// TIA Portal V20 export
FUNCTION_BLOCK "LER_Axis"   // FB60, LAD
// stored: Access Published, MemoryReserve 100, Namespace Homing, SetENOAutomatically false
   VAR_INPUT
      Status : "LAF_typeUnitStatus";
      HMI : Bool;
      Process : Bool;
      int1 { ExternalAccessible := 'False'; ExternalVisible := 'False'; ExternalWritable := 'False'} : Bool := true;
      int2 { ExternalAccessible := 'False'; ExternalVisible := 'False'; ExternalWritable := 'False'} : Bool := true;
      int3 { ExternalAccessible := 'False'; ExternalVisible := 'False'; ExternalWritable := 'False'} : Bool := true;
      int4 { ExternalAccessible := 'False'; ExternalVisible := 'False'; ExternalWritable := 'False'} : Bool := true;
      int5 { ExternalAccessible := 'False'; ExternalVisible := 'False'; ExternalWritable := 'False'} : Bool := true;
      int6 { ExternalAccessible := 'False'; ExternalVisible := 'False'; ExternalWritable := 'False'} : Bool := true;
      int7 { ExternalAccessible := 'False'; ExternalVisible := 'False'; ExternalWritable := 'False'} : Bool := true;
      int8 { ExternalAccessible := 'False'; ExternalVisible := 'False'; ExternalWritable := 'False'} : Bool := true;
      int9 { ExternalAccessible := 'False'; ExternalVisible := 'False'; ExternalWritable := 'False'} : Bool := true;
      int10 { ExternalAccessible := 'False'; ExternalVisible := 'False'; ExternalWritable := 'False'} : Bool := true;
      Bypass : Bool := true;
   END_VAR
   VAR_OUTPUT
      HomeInterlock : Bool;
   END_VAR
   VAR_IN_OUT
      intout : Array[0..9] of Bool;
   END_VAR
   VAR
      HomeCondition : Bool;
      HomeNotCondition : Bool;
   END_VAR
BEGIN

REGION Network 2 (SCL)
       IF (#int1 AND #int2 AND #int3 AND #int4 AND #int5 AND #int6 AND #int7 AND #int8 AND #int9 AND #int10) OR #Bypass THEN
           #HomeCondition := TRUE;
           #HomeNotCondition := FALSE;


           IF #HMI OR #Process THEN
               #intout[0] := FALSE;
               #intout[1] := FALSE;
               #intout[2] := FALSE;
               #intout[3] := FALSE;
               #intout[4] := FALSE;
               #intout[5] := FALSE;
               #intout[6] := FALSE;
               #intout[7] := FALSE;
               #intout[8] := FALSE;
               #intout[9] := FALSE;
           END_IF;


    ELSE
               #HomeCondition := FALSE;
               #HomeNotCondition := TRUE;

           IF #HMI OR #Process THEN

               IF NOT #int1 THEN
                   #intout[0] := TRUE;
               ELSE
                   #intout[0] := FALSE;
               END_IF;
               IF NOT #int2 THEN
                   #intout[1] := TRUE;
               ELSE
                   #intout[1] := FALSE;
               END_IF;
               IF NOT #int3 THEN
                   #intout[2] := TRUE;
               ELSE
                   #intout[2] := FALSE;
               END_IF;
               IF NOT #int4 THEN
                   #intout[3] := TRUE;
               ELSE
                   #intout[3] := FALSE;
               END_IF;
               IF NOT #int5 THEN
                   #intout[4] := TRUE;
               ELSE
                   #intout[4] := FALSE;
               END_IF;
               IF NOT #int6 THEN
                   #intout[5] := TRUE;
               ELSE
                   #intout[5] := FALSE;
               END_IF;
               IF NOT #int7 THEN
                   #intout[6] := TRUE;
               ELSE
                   #intout[6] := FALSE;
               END_IF;
               IF NOT #int8 THEN
                   #intout[7] := TRUE;
               ELSE
                   #intout[7] := FALSE;
               END_IF;
               IF NOT #int9 THEN
                   #intout[8] := TRUE;
               ELSE
                   #intout[8] := FALSE;
               END_IF;
               IF NOT #int10 THEN
                   #intout[9] := TRUE;
               ELSE
                   #intout[9] := FALSE;
               END_IF;

           END_IF;

       END_IF;
       #HomeInterlock := #HomeCondition;
END_REGION
END_FUNCTION_BLOCK
